// SIMATIC S7-200 project (STEP 7-Micro/WIN), CPU 224 CN REL 02.01

ORGANIZATION_BLOCK MAIN:OB1
TITLE=程序注释
BEGIN
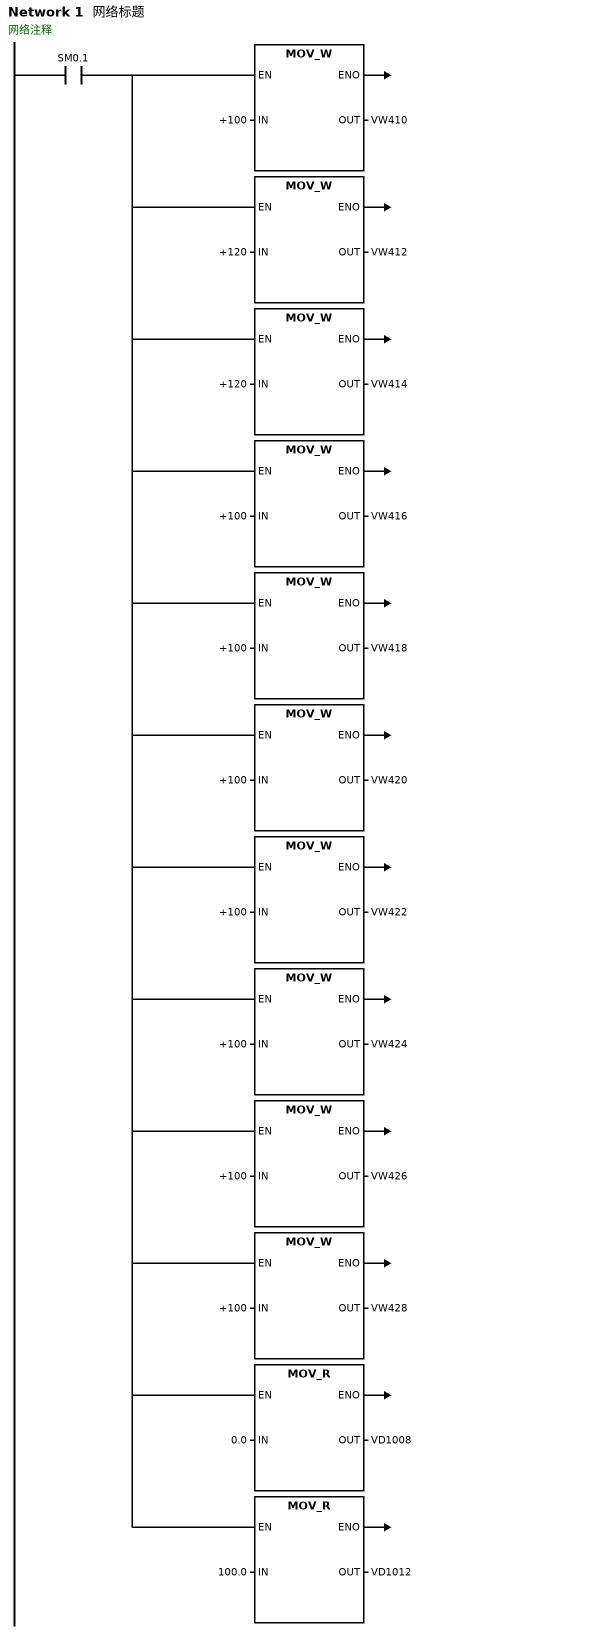
Network 1 // 网络标题
// 网络注释
LD     SM0.1
MOVW   +100, VW410
MOVW   +120, VW412
MOVW   +120, VW414
MOVW   +100, VW416
MOVW   +100, VW418
MOVW   +100, VW420
MOVW   +100, VW422
MOVW   +100, VW424
MOVW   +100, VW426
MOVW   +100, VW428
MOVR   0.0, VD1008
MOVR   100.0, VD1012
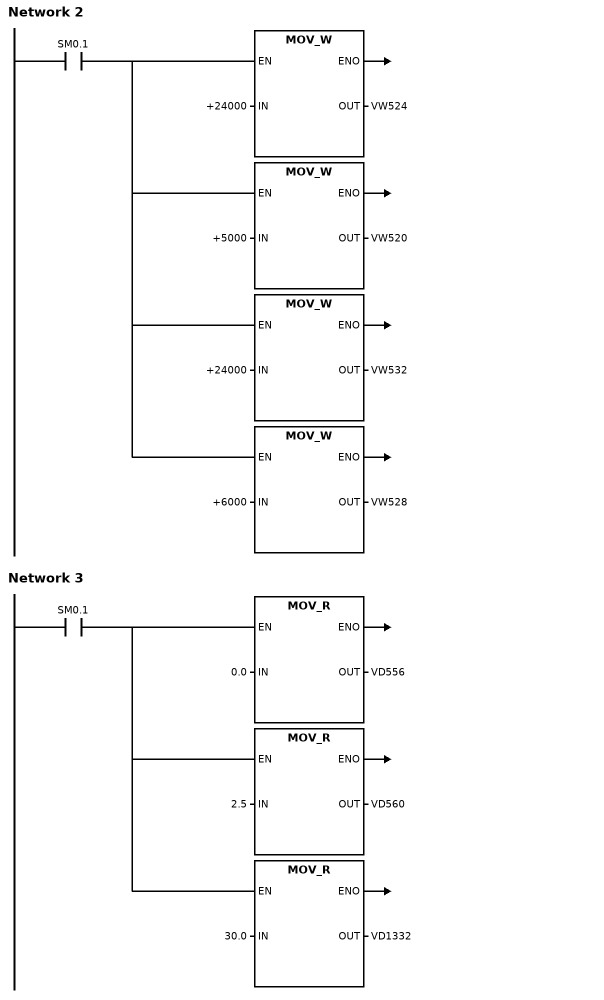
Network 2
LD     SM0.1
MOVW   +24000, VW524
MOVW   +5000, VW520
MOVW   +24000, VW532
MOVW   +6000, VW528
Network 3
LD     SM0.1
MOVR   0.0, VD556
MOVR   2.5, VD560
MOVR   30.0, VD1332
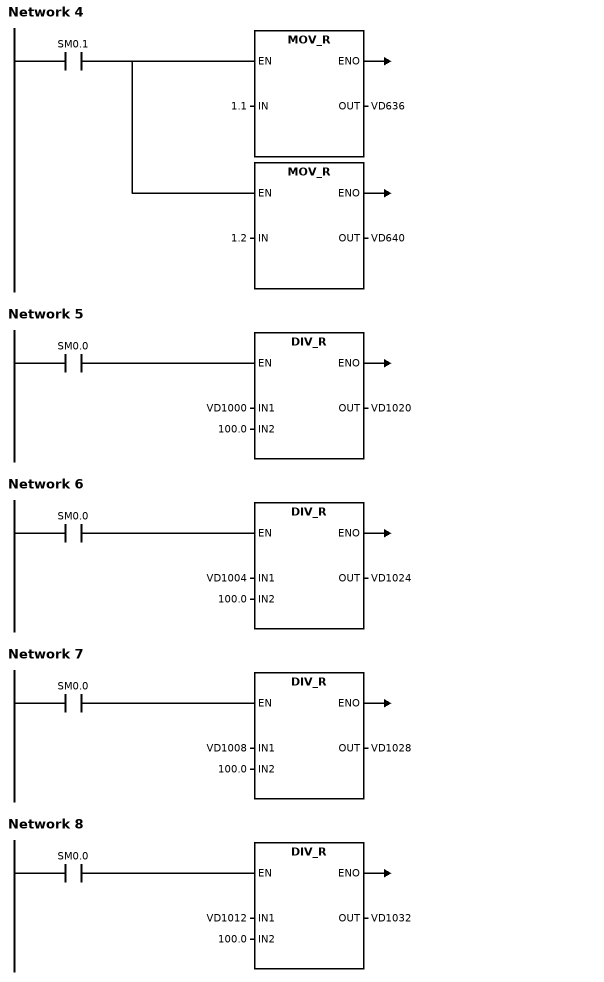
Network 4
LD     SM0.1
MOVR   1.1, VD636
MOVR   1.2, VD640
Network 5
LD     SM0.0
MOVR   VD1000, VD1020
/R     100.0, VD1020
Network 6
LD     SM0.0
MOVR   VD1004, VD1024
/R     100.0, VD1024
Network 7
LD     SM0.0
MOVR   VD1008, VD1028
/R     100.0, VD1028
Network 8
LD     SM0.0
MOVR   VD1012, VD1032
/R     100.0, VD1032
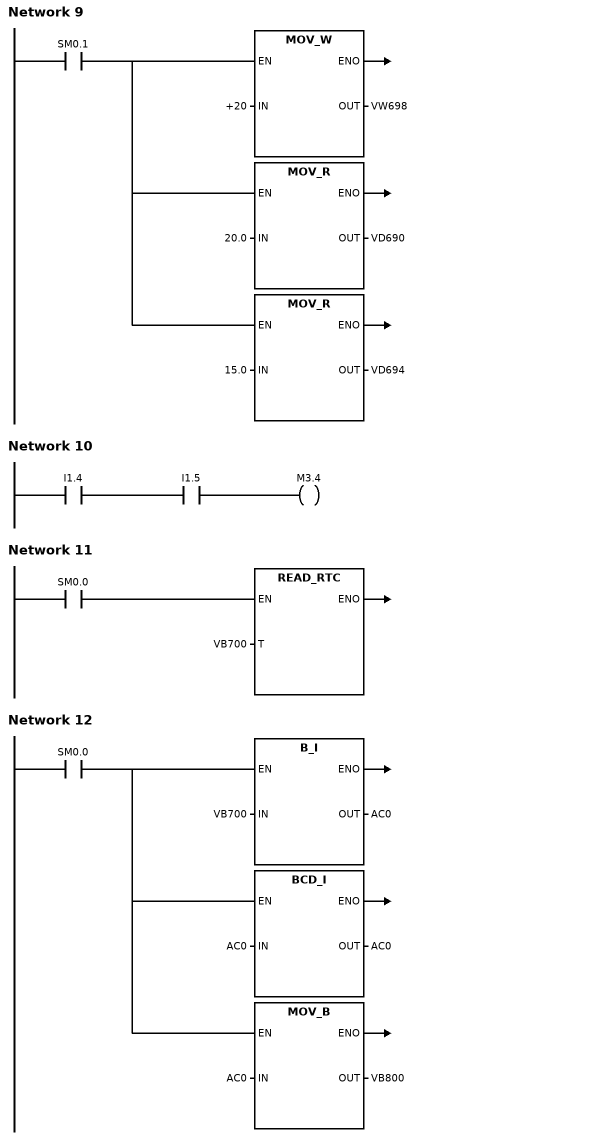
Network 9
LD     SM0.1
MOVW   +20, VW698
MOVR   20.0, VD690
MOVR   15.0, VD694
Network 10
LD     I1.4
A      I1.5
=      M3.4
Network 11
LD     SM0.0
TODR   VB700
Network 12
LD     SM0.0
BTI    VB700, AC0
BCDI   AC0
MOVB   AC0, VB800
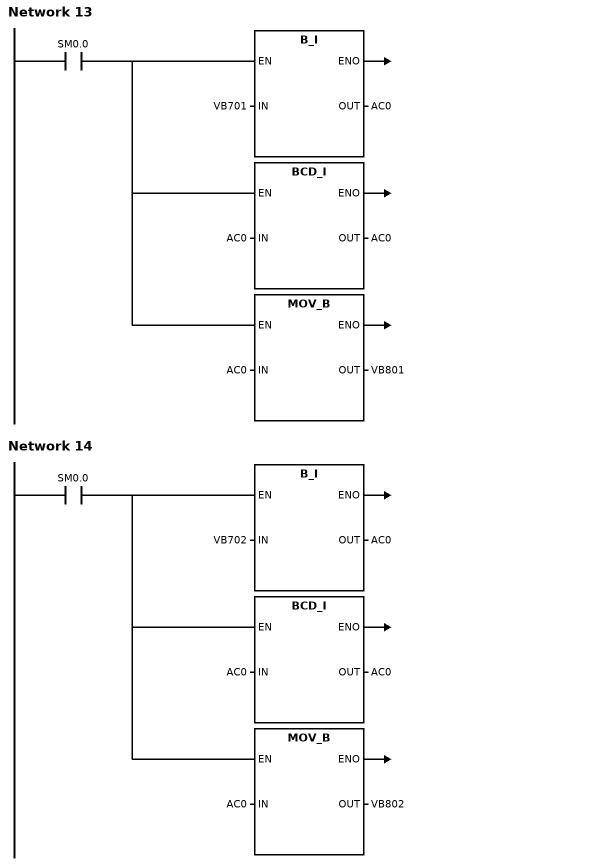
Network 13
LD     SM0.0
BTI    VB701, AC0
BCDI   AC0
MOVB   AC0, VB801
Network 14
LD     SM0.0
BTI    VB702, AC0
BCDI   AC0
MOVB   AC0, VB802
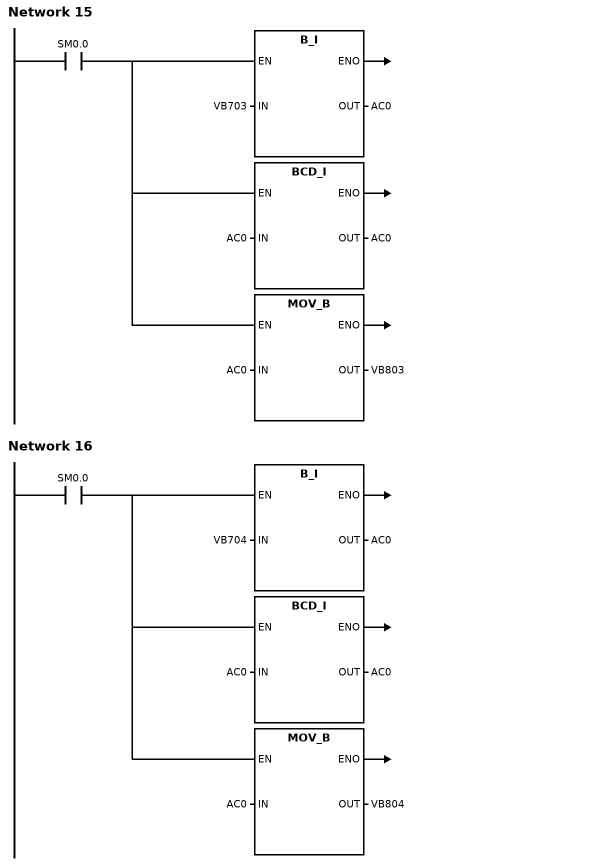
Network 15
LD     SM0.0
BTI    VB703, AC0
BCDI   AC0
MOVB   AC0, VB803
Network 16
LD     SM0.0
BTI    VB704, AC0
BCDI   AC0
MOVB   AC0, VB804
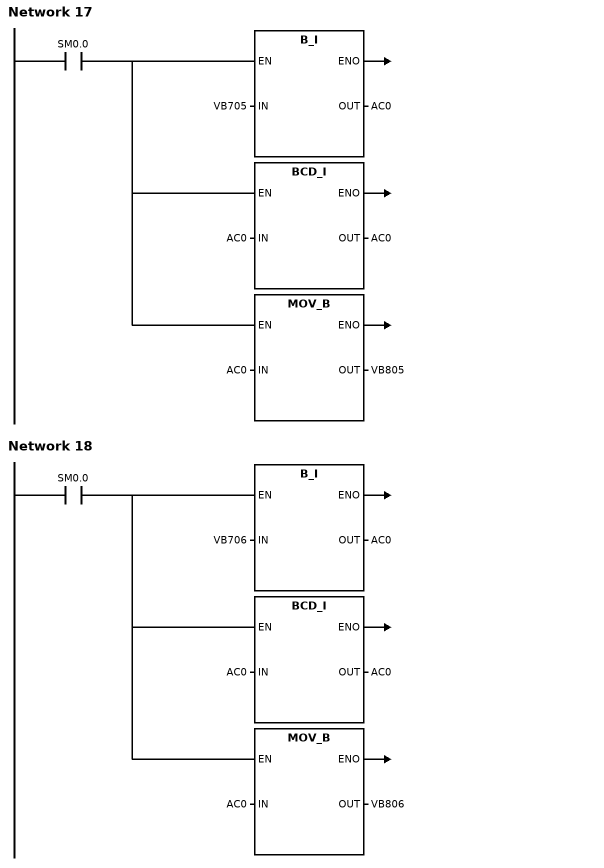
Network 17
LD     SM0.0
BTI    VB705, AC0
BCDI   AC0
MOVB   AC0, VB805
Network 18
LD     SM0.0
BTI    VB706, AC0
BCDI   AC0
MOVB   AC0, VB806
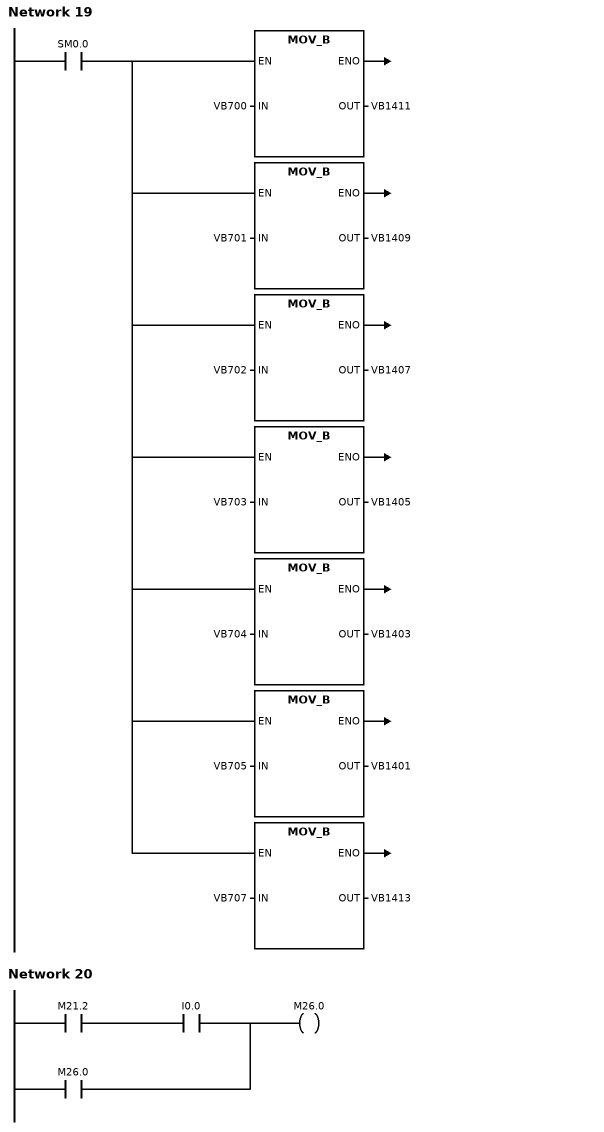
Network 19
LD     SM0.0
MOVB   VB700, VB1411
MOVB   VB701, VB1409
MOVB   VB702, VB1407
MOVB   VB703, VB1405
MOVB   VB704, VB1403
MOVB   VB705, VB1401
MOVB   VB707, VB1413
Network 20
LD     M21.2
A      I0.0
O      M26.0
=      M26.0
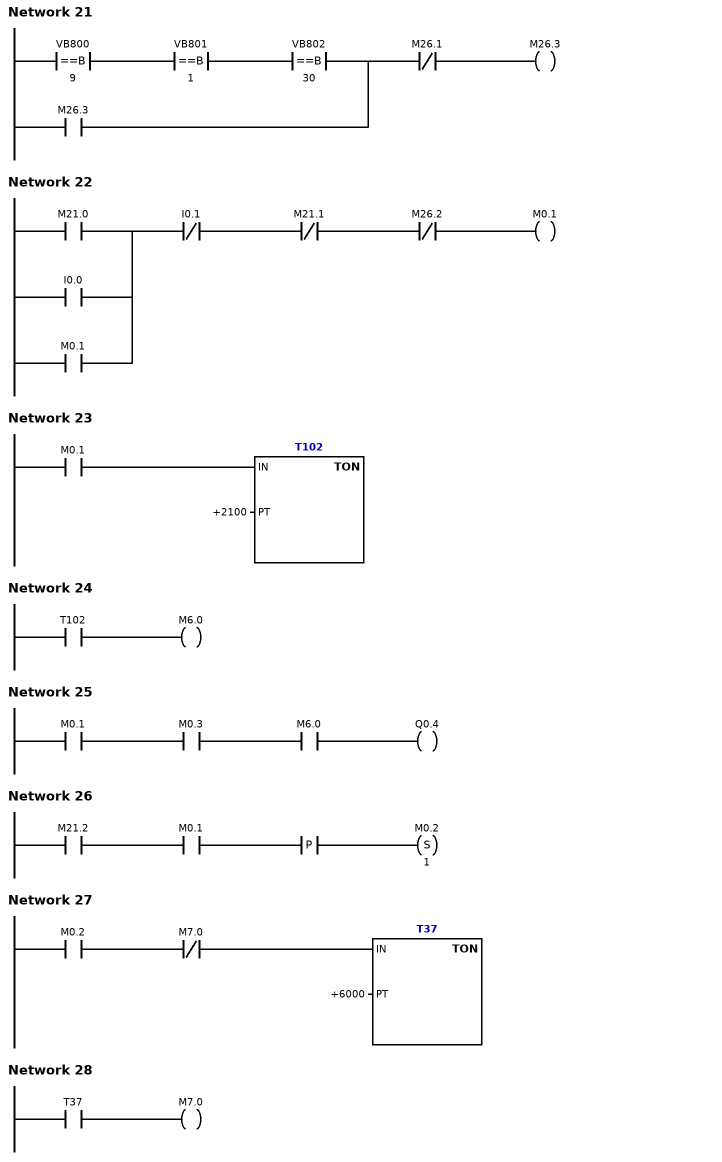
Network 21
LDB=   VB800, 9
AB=    VB801, 1
AB=    VB802, 30
O      M26.3
AN     M26.1
=      M26.3
Network 22
LD     M21.0
O      I0.0
O      M0.1
AN     I0.1
AN     M21.1
AN     M26.2
=      M0.1
Network 23
LD     M0.1
TON    T102, +2100
Network 24
LD     T102
=      M6.0
Network 25
LD     M0.1
A      M0.3
A      M6.0
=      Q0.4
Network 26
LD     M21.2
A      M0.1
EU
S      M0.2, 1
Network 27
LD     M0.2
AN     M7.0
TON    T37, +6000
Network 28
LD     T37
=      M7.0
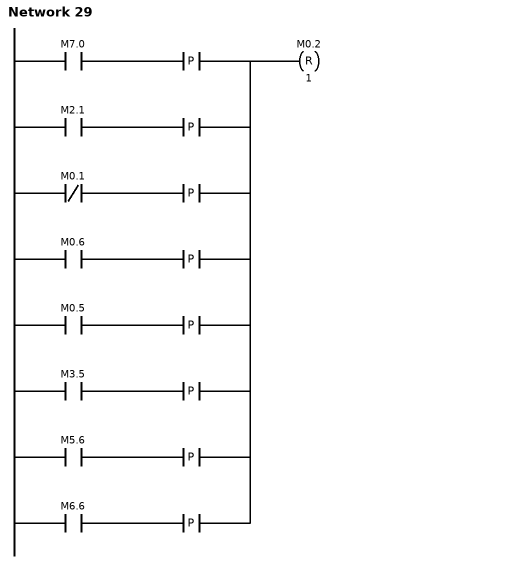
Network 29
LD     M7.0
EU
LD     M2.1
EU
OLD
LDN    M0.1
EU
OLD
LD     M0.6
EU
OLD
LD     M0.5
EU
OLD
LD     M3.5
EU
OLD
LD     M5.6
EU
OLD
LD     M6.6
EU
OLD
R      M0.2, 1
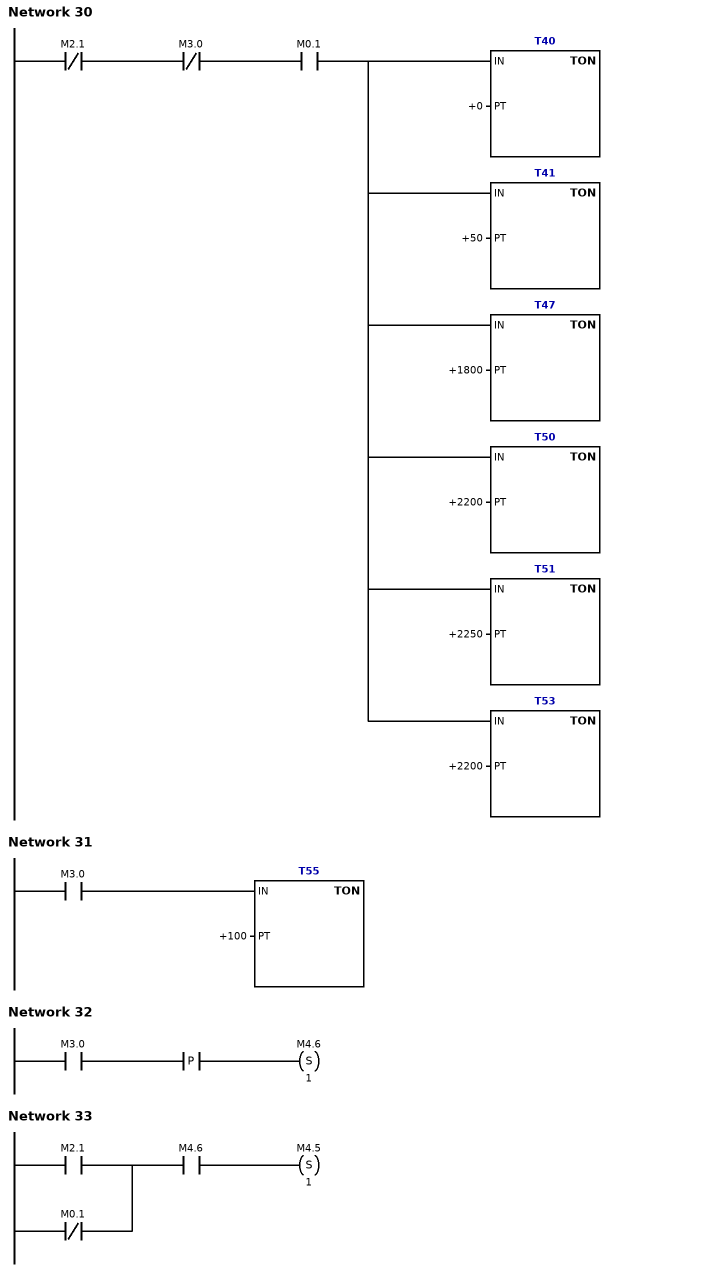
Network 30
LDN    M2.1
AN     M3.0
A      M0.1
TON    T40, +0
TON    T41, +50
TON    T47, +1800
TON    T50, +2200
TON    T51, +2250
TON    T53, +2200
Network 31
LD     M3.0
TON    T55, +100
Network 32
LD     M3.0
EU
S      M4.6, 1
Network 33
LD     M2.1
ON     M0.1
A      M4.6
S      M4.5, 1
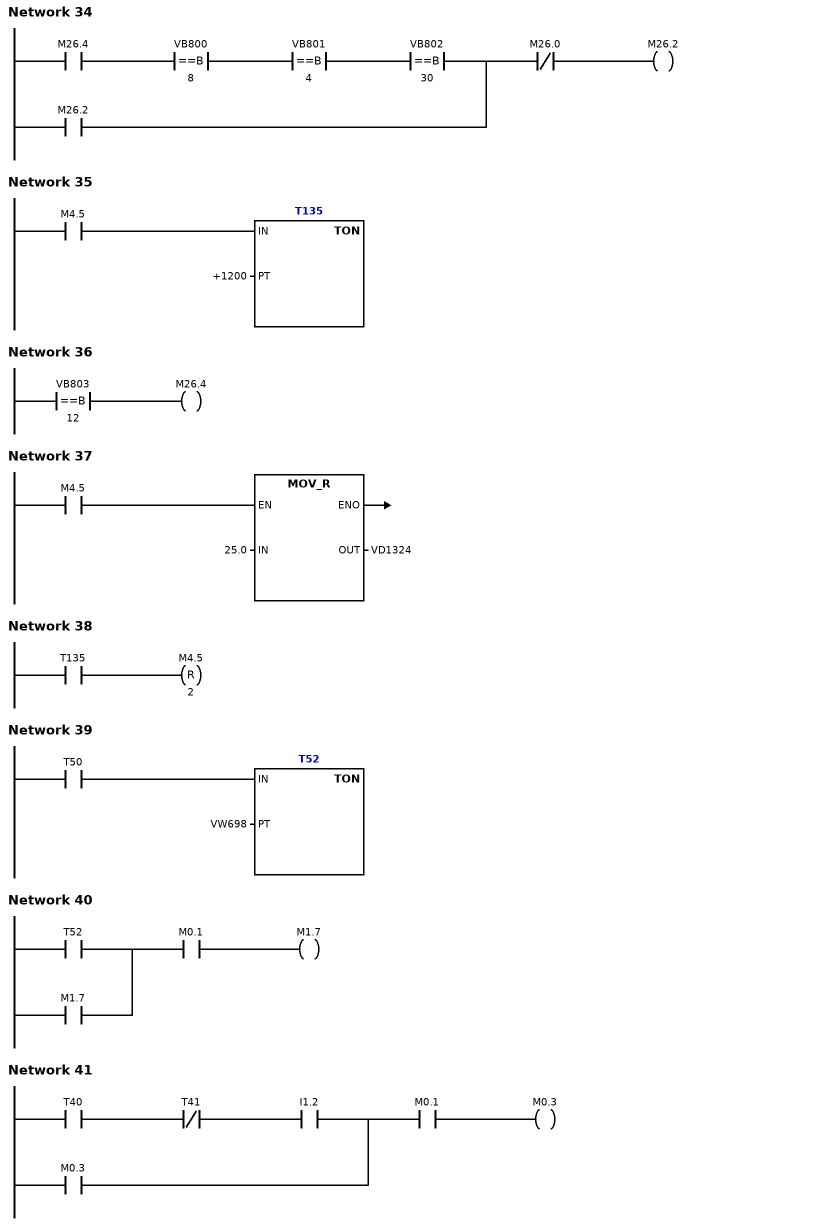
Network 34
LD     M26.4
AB=    VB800, 8
AB=    VB801, 4
AB=    VB802, 30
O      M26.2
AN     M26.0
=      M26.2
Network 35
LD     M4.5
TON    T135, +1200
Network 36
LDB=   VB803, 12
=      M26.4
Network 37
LD     M4.5
MOVR   25.0, VD1324
Network 38
LD     T135
R      M4.5, 2
Network 39
LD     T50
TON    T52, VW698
Network 40
LD     T52
O      M1.7
A      M0.1
=      M1.7
Network 41
LD     T40
AN     T41
A      I1.2
O      M0.3
A      M0.1
=      M0.3
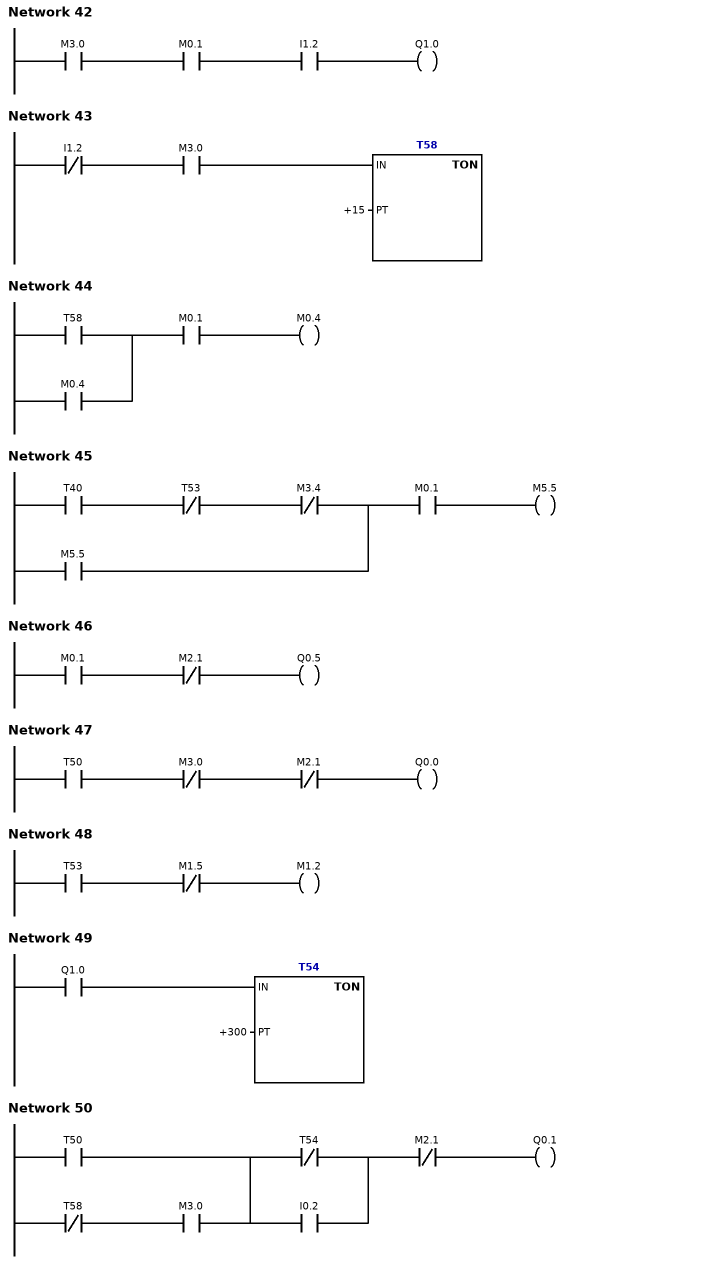
Network 42
LD     M3.0
A      M0.1
A      I1.2
=      Q1.0
Network 43
LDN    I1.2
A      M3.0
TON    T58, +15
Network 44
LD     T58
O      M0.4
A      M0.1
=      M0.4
Network 45
LD     T40
AN     T53
AN     M3.4
O      M5.5
A      M0.1
=      M5.5
Network 46
LD     M0.1
AN     M2.1
=      Q0.5
Network 47
LD     T50
AN     M3.0
AN     M2.1
=      Q0.0
Network 48
LD     T53
AN     M1.5
=      M1.2
Network 49
LD     Q1.0
TON    T54, +300
Network 50
LD     T50
LDN    T58
A      M3.0
OLD
LDN    T54
O      I0.2
ALD
AN     M2.1
=      Q0.1
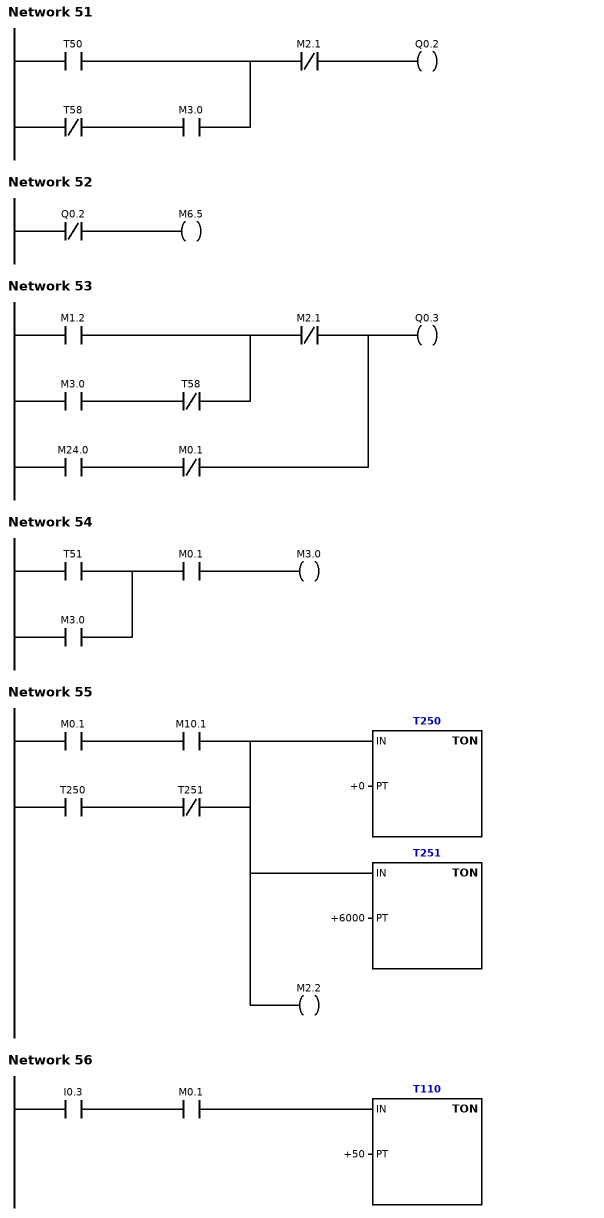
Network 51
LD     T50
LDN    T58
A      M3.0
OLD
AN     M2.1
=      Q0.2
Network 52
LDN    Q0.2
=      M6.5
Network 53
LD     M1.2
LD     M3.0
AN     T58
OLD
AN     M2.1
LD     M24.0
AN     M0.1
OLD
=      Q0.3
Network 54
LD     T51
O      M3.0
A      M0.1
=      M3.0
Network 55
LD     M0.1
A      M10.1
LD     T250
AN     T251
OLD
TON    T250, +0
TON    T251, +6000
=      M2.2
Network 56
LD     I0.3
A      M0.1
TON    T110, +50
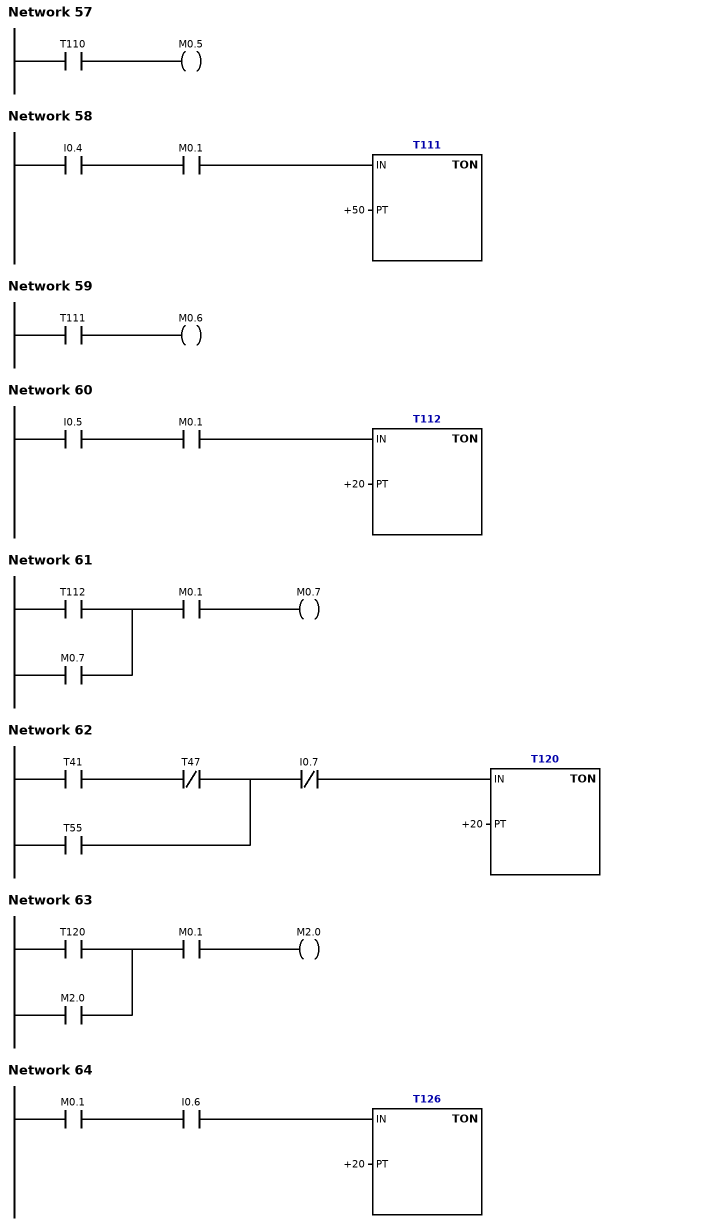
Network 57
LD     T110
=      M0.5
Network 58
LD     I0.4
A      M0.1
TON    T111, +50
Network 59
LD     T111
=      M0.6
Network 60
LD     I0.5
A      M0.1
TON    T112, +20
Network 61
LD     T112
O      M0.7
A      M0.1
=      M0.7
Network 62
LD     T41
AN     T47
O      T55
AN     I0.7
TON    T120, +20
Network 63
LD     T120
O      M2.0
A      M0.1
=      M2.0
Network 64
LD     M0.1
A      I0.6
TON    T126, +20
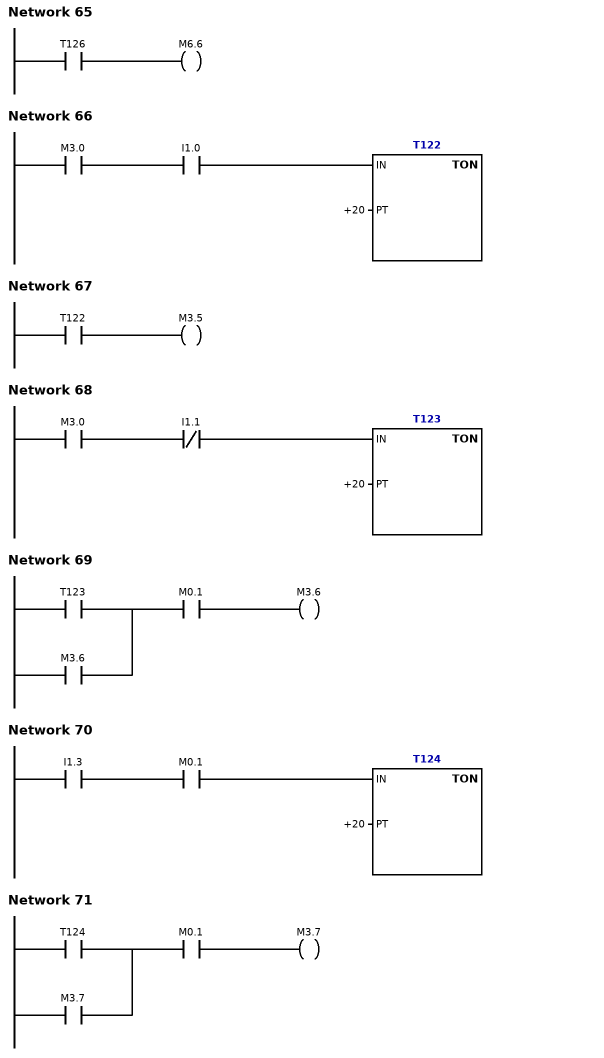
Network 65
LD     T126
=      M6.6
Network 66
LD     M3.0
A      I1.0
TON    T122, +20
Network 67
LD     T122
=      M3.5
Network 68
LD     M3.0
AN     I1.1
TON    T123, +20
Network 69
LD     T123
O      M3.6
A      M0.1
=      M3.6
Network 70
LD     I1.3
A      M0.1
TON    T124, +20
Network 71
LD     T124
O      M3.7
A      M0.1
=      M3.7
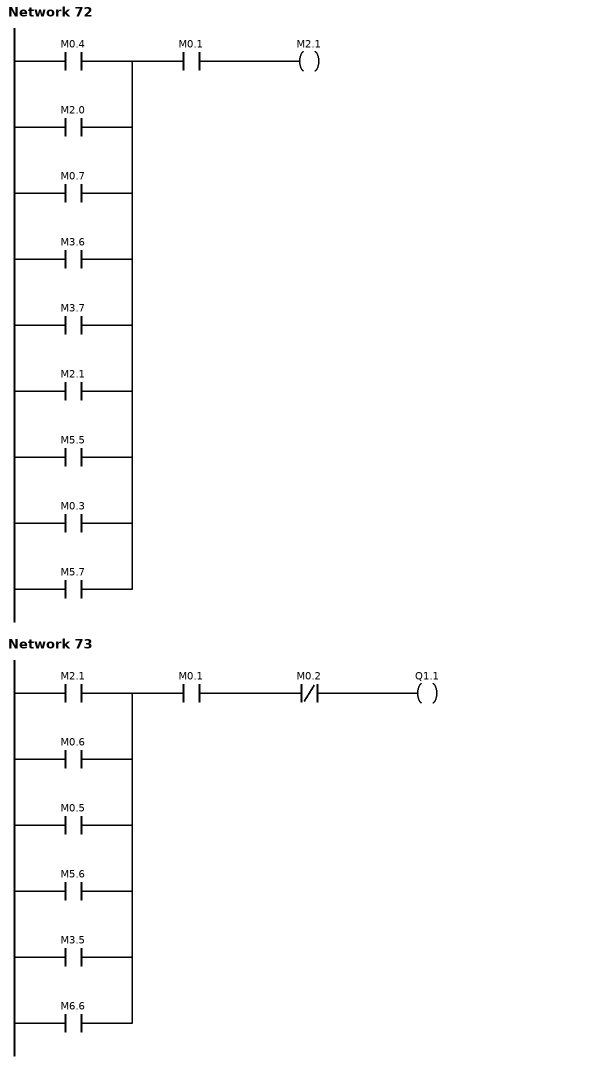
Network 72
LD     M0.4
O      M2.0
O      M0.7
O      M3.6
O      M3.7
O      M2.1
O      M5.5
O      M0.3
O      M5.7
A      M0.1
=      M2.1
Network 73
LD     M2.1
O      M0.6
O      M0.5
O      M5.6
O      M3.5
O      M6.6
A      M0.1
AN     M0.2
=      Q1.1
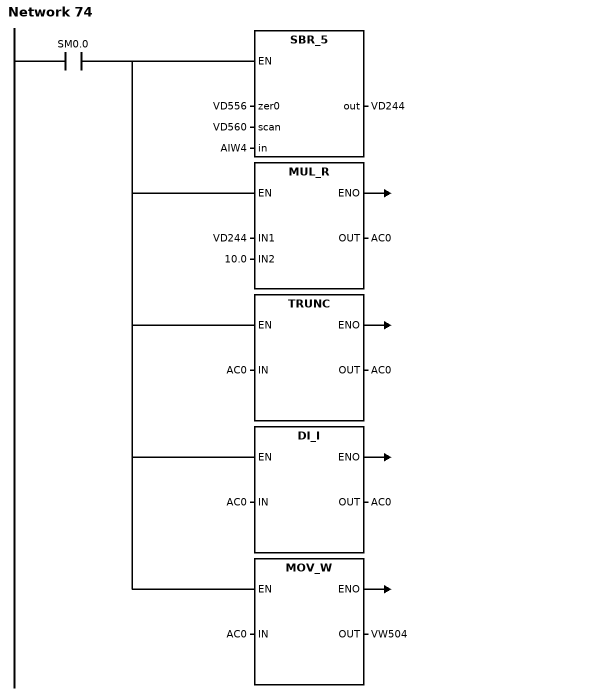
Network 74
LD     SM0.0
CALL   SBR_5:SBR5, VD556, VD560, AIW4, VD244
MOVR   VD244, AC0
*R     10.0, AC0
TRUNC  AC0, AC0
DTI    AC0, AC0
MOVW   AC0, VW504
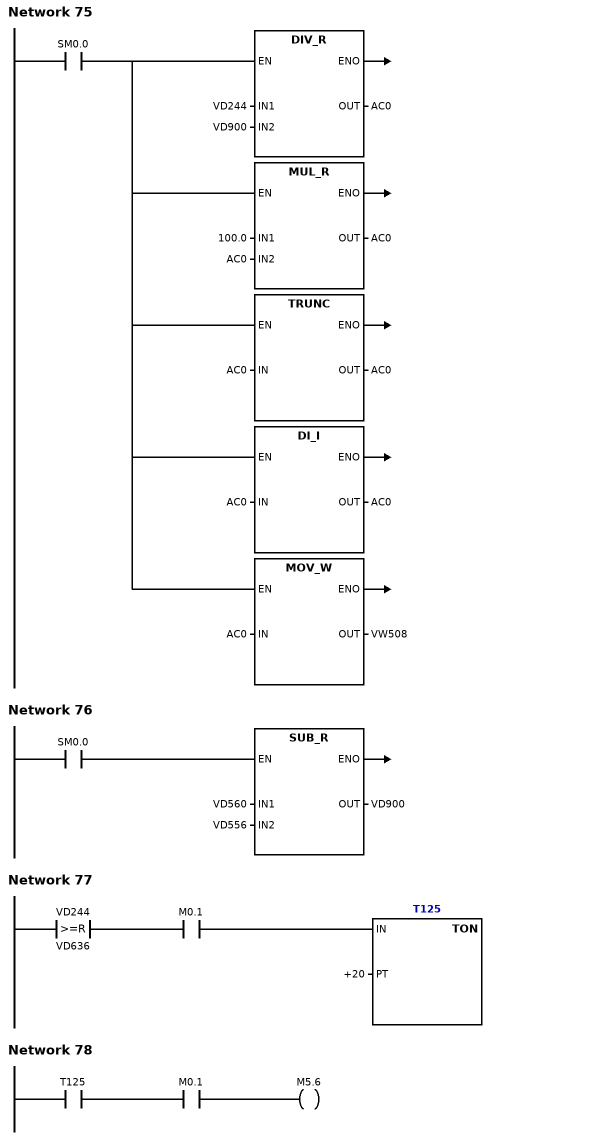
Network 75
LD     SM0.0
MOVR   VD244, AC0
/R     VD900, AC0
*R     100.0, AC0
TRUNC  AC0, AC0
DTI    AC0, AC0
MOVW   AC0, VW508
Network 76
LD     SM0.0
MOVR   VD560, VD900
-R     VD556, VD900
Network 77
LDR>=  VD244, VD636
A      M0.1
TON    T125, +20
Network 78
LD     T125
A      M0.1
=      M5.6
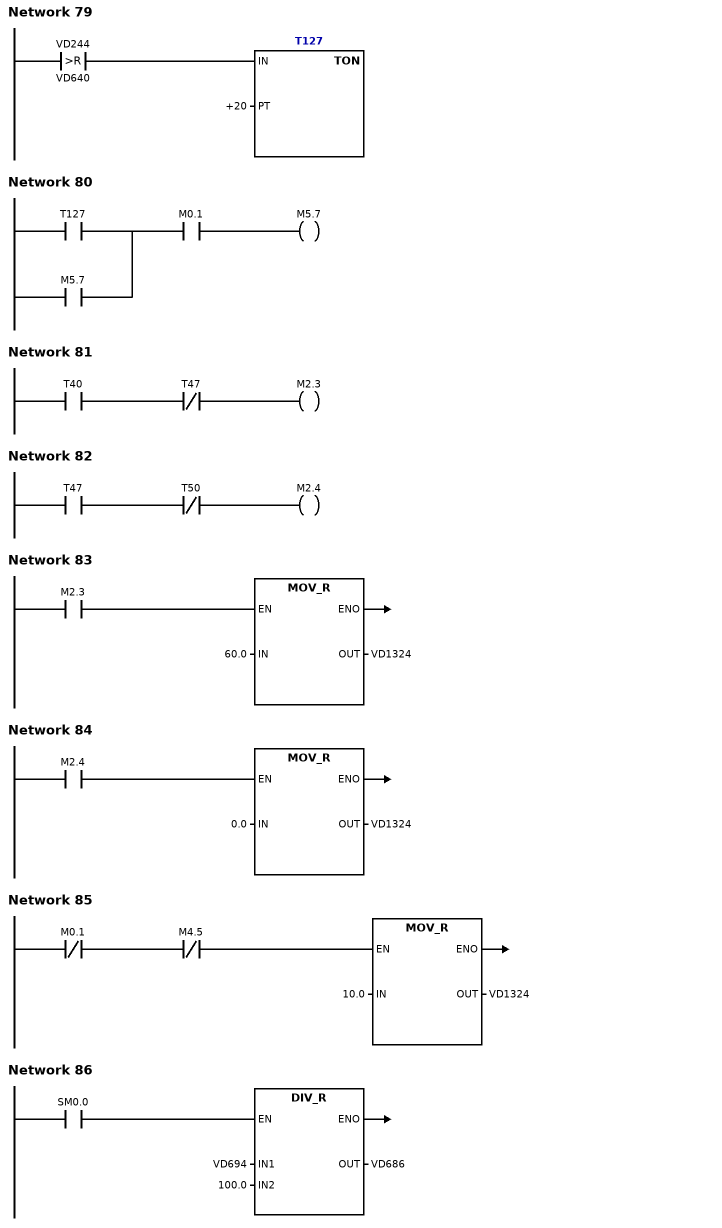
Network 79
LDR>   VD244, VD640
TON    T127, +20
Network 80
LD     T127
O      M5.7
A      M0.1
=      M5.7
Network 81
LD     T40
AN     T47
=      M2.3
Network 82
LD     T47
AN     T50
=      M2.4
Network 83
LD     M2.3
MOVR   60.0, VD1324
Network 84
LD     M2.4
MOVR   0.0, VD1324
Network 85
LDN    M0.1
AN     M4.5
MOVR   10.0, VD1324
Network 86
LD     SM0.0
MOVR   VD694, VD686
/R     100.0, VD686
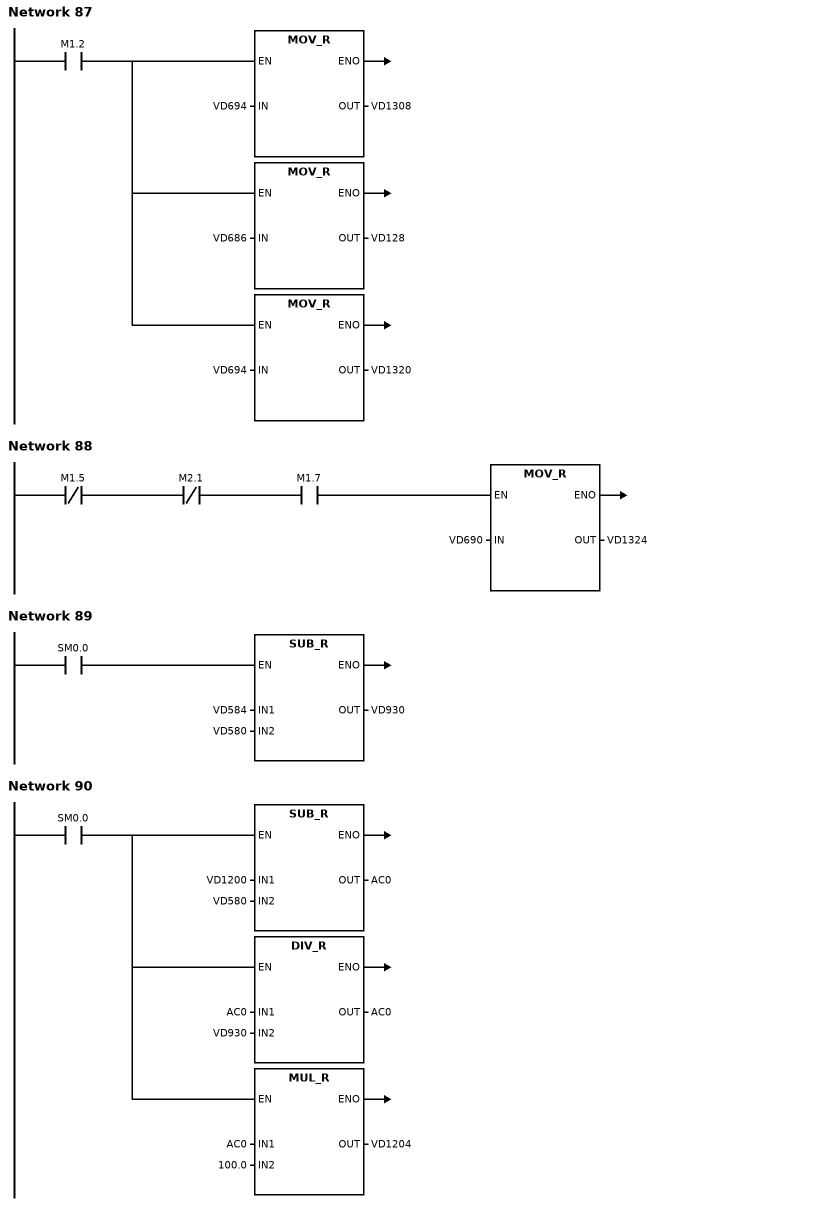
Network 87
LD     M1.2
MOVR   VD694, VD1308
MOVR   VD686, VD128
MOVR   VD694, VD1320
Network 88
LDN    M1.5
AN     M2.1
A      M1.7
MOVR   VD690, VD1324
Network 89
LD     SM0.0
MOVR   VD584, VD930
-R     VD580, VD930
Network 90
LD     SM0.0
MOVR   VD1200, AC0
-R     VD580, AC0
/R     VD930, AC0
MOVR   AC0, VD1204
*R     100.0, VD1204
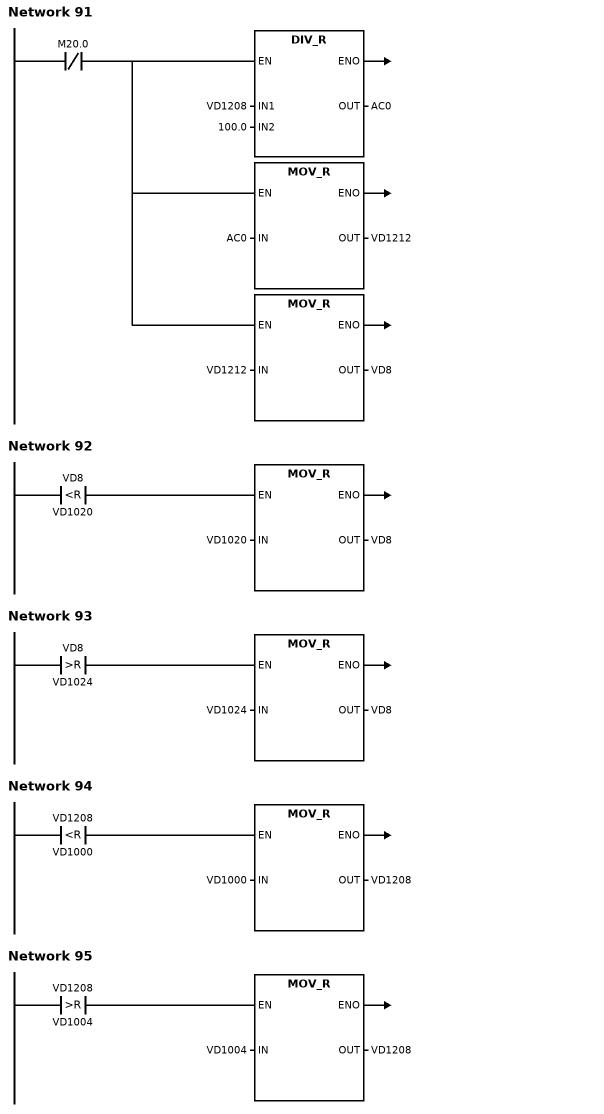
Network 91
LDN    M20.0
MOVR   VD1208, AC0
/R     100.0, AC0
MOVR   AC0, VD1212
MOVR   VD1212, VD8
Network 92
LDR<   VD8, VD1020
MOVR   VD1020, VD8
Network 93
LDR>   VD8, VD1024
MOVR   VD1024, VD8
Network 94
LDR<   VD1208, VD1000
MOVR   VD1000, VD1208
Network 95
LDR>   VD1208, VD1004
MOVR   VD1004, VD1208
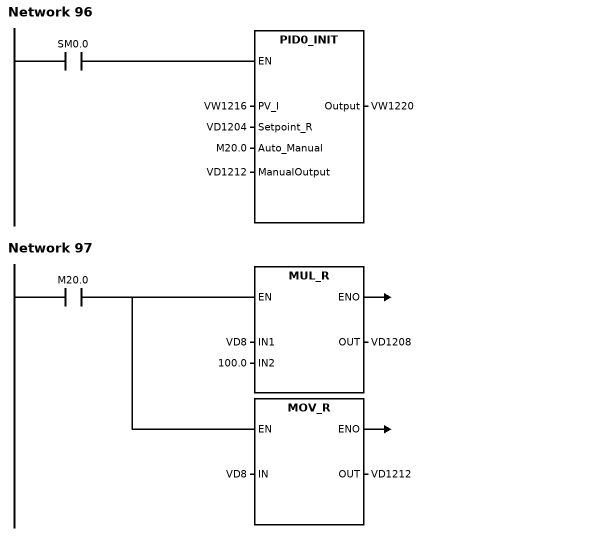
Network 96
LD     SM0.0
CALL   PID0_INIT:SBR1, VW1216, VD1204, M20.0, VD1212, VW1220
Network 97
LD     M20.0
MOVR   VD8, VD1208
*R     100.0, VD1208
MOVR   VD8, VD1212
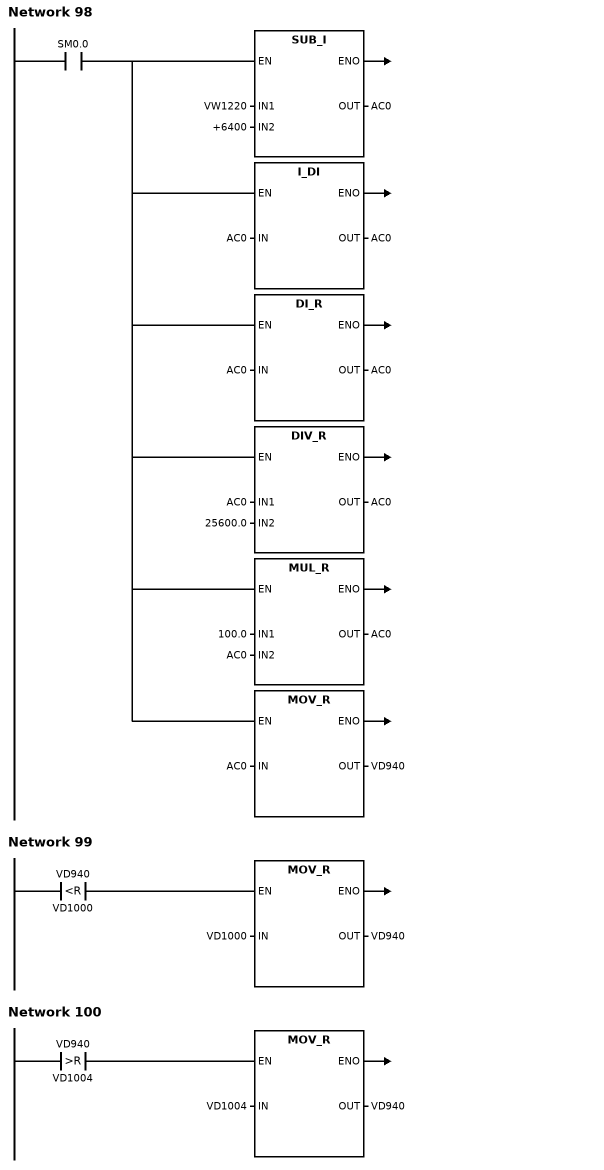
Network 98
LD     SM0.0
MOVW   VW1220, AC0
-I     +6400, AC0
ITD    AC0, AC0
DTR    AC0, AC0
/R     25600.0, AC0
*R     100.0, AC0
MOVR   AC0, VD940
Network 99
LDR<   VD940, VD1000
MOVR   VD1000, VD940
Network 100
LDR>   VD940, VD1004
MOVR   VD1004, VD940
